TYPE EL1809_PDOS :
	STRUCT
		
		HwToPLC : EL1809_HWTOPLC_PDOS;
		
	END_STRUCT
END_TYPE

(* stored: Version 1.1.0.1
   DUT EL1809_PDOS: Id {6667a0d9-4c36-4afe-94e3-3b411804f9a2} *)
